FUNCTION_BLOCK ASSEMBLE_AD_FROM_AX (* this Function combines the 32 AX (BOOL) adapters to a AD (DWORD) *)
  (* Standard: 61499-2; Description: Copyright (c) 2026 Meisterschulen am Ostbahnhof SPDX-License-Identifier: EPL-2.0 *)
  (* Version 1.0, 2026-05-16, Franz Höpfinger, Meisterschulen am Ostbahnhof, initial API and implementation and/or initial documentation *)
  PACKAGE adapter::assembling;
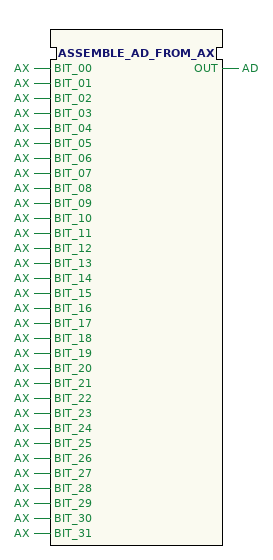
  SOCKETS
    BIT_00 : adapter::types::unidirectional::AX; (* Bool Bit 0 *)
    BIT_01 : adapter::types::unidirectional::AX; (* Bool Bit 1 *)
    BIT_02 : adapter::types::unidirectional::AX; (* Bool Bit 2 *)
    BIT_03 : adapter::types::unidirectional::AX; (* Bool Bit 3 *)
    BIT_04 : adapter::types::unidirectional::AX; (* Bool Bit 4 *)
    BIT_05 : adapter::types::unidirectional::AX; (* Bool Bit 5 *)
    BIT_06 : adapter::types::unidirectional::AX; (* Bool Bit 6 *)
    BIT_07 : adapter::types::unidirectional::AX; (* Bool Bit 7 *)
    BIT_08 : adapter::types::unidirectional::AX; (* Bool Bit 8 *)
    BIT_09 : adapter::types::unidirectional::AX; (* Bool Bit 9 *)
    BIT_10 : adapter::types::unidirectional::AX; (* Bool Bit 10 *)
    BIT_11 : adapter::types::unidirectional::AX; (* Bool Bit 11 *)
    BIT_12 : adapter::types::unidirectional::AX; (* Bool Bit 12 *)
    BIT_13 : adapter::types::unidirectional::AX; (* Bool Bit 13 *)
    BIT_14 : adapter::types::unidirectional::AX; (* Bool Bit 14 *)
    BIT_15 : adapter::types::unidirectional::AX; (* Bool Bit 15 *)
    BIT_16 : adapter::types::unidirectional::AX; (* Bool Bit 16 *)
    BIT_17 : adapter::types::unidirectional::AX; (* Bool Bit 17 *)
    BIT_18 : adapter::types::unidirectional::AX; (* Bool Bit 18 *)
    BIT_19 : adapter::types::unidirectional::AX; (* Bool Bit 19 *)
    BIT_20 : adapter::types::unidirectional::AX; (* Bool Bit 20 *)
    BIT_21 : adapter::types::unidirectional::AX; (* Bool Bit 21 *)
    BIT_22 : adapter::types::unidirectional::AX; (* Bool Bit 22 *)
    BIT_23 : adapter::types::unidirectional::AX; (* Bool Bit 23 *)
    BIT_24 : adapter::types::unidirectional::AX; (* Bool Bit 24 *)
    BIT_25 : adapter::types::unidirectional::AX; (* Bool Bit 25 *)
    BIT_26 : adapter::types::unidirectional::AX; (* Bool Bit 26 *)
    BIT_27 : adapter::types::unidirectional::AX; (* Bool Bit 27 *)
    BIT_28 : adapter::types::unidirectional::AX; (* Bool Bit 28 *)
    BIT_29 : adapter::types::unidirectional::AX; (* Bool Bit 29 *)
    BIT_30 : adapter::types::unidirectional::AX; (* Bool Bit 30 *)
    BIT_31 : adapter::types::unidirectional::AX; (* Bool Bit 31 *)
  END_SOCKETS
  PLUGS
    OUT : adapter::types::unidirectional::AD; (* DWORD Output *)
  END_PLUGS
  FBS
    ASSEMBLE_DWORD_FROM_BOOLS : eclipse4diac::utils::assembling::ASSEMBLE_DWORD_FROM_BOOLS;
    E_D_FF_ANY : iec61499::events::E_D_FF_ANY;
  END_FBS
  EVENT_CONNECTIONS
    BIT_00.E1 TO ASSEMBLE_DWORD_FROM_BOOLS.REQ;
    BIT_01.E1 TO ASSEMBLE_DWORD_FROM_BOOLS.REQ;
    BIT_02.E1 TO ASSEMBLE_DWORD_FROM_BOOLS.REQ;
    BIT_03.E1 TO ASSEMBLE_DWORD_FROM_BOOLS.REQ;
    BIT_04.E1 TO ASSEMBLE_DWORD_FROM_BOOLS.REQ;
    BIT_05.E1 TO ASSEMBLE_DWORD_FROM_BOOLS.REQ;
    BIT_06.E1 TO ASSEMBLE_DWORD_FROM_BOOLS.REQ;
    BIT_07.E1 TO ASSEMBLE_DWORD_FROM_BOOLS.REQ;
    BIT_08.E1 TO ASSEMBLE_DWORD_FROM_BOOLS.REQ;
    BIT_09.E1 TO ASSEMBLE_DWORD_FROM_BOOLS.REQ;
    BIT_10.E1 TO ASSEMBLE_DWORD_FROM_BOOLS.REQ;
    BIT_11.E1 TO ASSEMBLE_DWORD_FROM_BOOLS.REQ;
    BIT_12.E1 TO ASSEMBLE_DWORD_FROM_BOOLS.REQ;
    BIT_13.E1 TO ASSEMBLE_DWORD_FROM_BOOLS.REQ;
    BIT_14.E1 TO ASSEMBLE_DWORD_FROM_BOOLS.REQ;
    BIT_15.E1 TO ASSEMBLE_DWORD_FROM_BOOLS.REQ;
    BIT_16.E1 TO ASSEMBLE_DWORD_FROM_BOOLS.REQ;
    BIT_17.E1 TO ASSEMBLE_DWORD_FROM_BOOLS.REQ;
    BIT_18.E1 TO ASSEMBLE_DWORD_FROM_BOOLS.REQ;
    BIT_19.E1 TO ASSEMBLE_DWORD_FROM_BOOLS.REQ;
    BIT_20.E1 TO ASSEMBLE_DWORD_FROM_BOOLS.REQ;
    BIT_21.E1 TO ASSEMBLE_DWORD_FROM_BOOLS.REQ;
    BIT_22.E1 TO ASSEMBLE_DWORD_FROM_BOOLS.REQ;
    BIT_23.E1 TO ASSEMBLE_DWORD_FROM_BOOLS.REQ;
    BIT_24.E1 TO ASSEMBLE_DWORD_FROM_BOOLS.REQ;
    BIT_25.E1 TO ASSEMBLE_DWORD_FROM_BOOLS.REQ;
    BIT_26.E1 TO ASSEMBLE_DWORD_FROM_BOOLS.REQ;
    BIT_27.E1 TO ASSEMBLE_DWORD_FROM_BOOLS.REQ;
    BIT_28.E1 TO ASSEMBLE_DWORD_FROM_BOOLS.REQ;
    BIT_29.E1 TO ASSEMBLE_DWORD_FROM_BOOLS.REQ;
    BIT_30.E1 TO ASSEMBLE_DWORD_FROM_BOOLS.REQ;
    BIT_31.E1 TO ASSEMBLE_DWORD_FROM_BOOLS.REQ;
    ASSEMBLE_DWORD_FROM_BOOLS.CNF TO E_D_FF_ANY.CLK;
    E_D_FF_ANY.EO TO OUT.E1;
  END_CONNECTIONS
  DATA_CONNECTIONS
    ASSEMBLE_DWORD_FROM_BOOLS. TO E_D_FF_ANY.D;
    E_D_FF_ANY.Q TO OUT.D1;
    BIT_31.D1 TO ASSEMBLE_DWORD_FROM_BOOLS.BIT_31;
    BIT_30.D1 TO ASSEMBLE_DWORD_FROM_BOOLS.BIT_30;
    BIT_29.D1 TO ASSEMBLE_DWORD_FROM_BOOLS.BIT_29;
    BIT_28.D1 TO ASSEMBLE_DWORD_FROM_BOOLS.BIT_28;
    BIT_27.D1 TO ASSEMBLE_DWORD_FROM_BOOLS.BIT_27;
    BIT_26.D1 TO ASSEMBLE_DWORD_FROM_BOOLS.BIT_26;
    BIT_25.D1 TO ASSEMBLE_DWORD_FROM_BOOLS.BIT_25;
    BIT_24.D1 TO ASSEMBLE_DWORD_FROM_BOOLS.BIT_24;
    BIT_23.D1 TO ASSEMBLE_DWORD_FROM_BOOLS.BIT_23;
    BIT_22.D1 TO ASSEMBLE_DWORD_FROM_BOOLS.BIT_22;
    BIT_21.D1 TO ASSEMBLE_DWORD_FROM_BOOLS.BIT_21;
    BIT_20.D1 TO ASSEMBLE_DWORD_FROM_BOOLS.BIT_20;
    BIT_19.D1 TO ASSEMBLE_DWORD_FROM_BOOLS.BIT_19;
    BIT_18.D1 TO ASSEMBLE_DWORD_FROM_BOOLS.BIT_18;
    BIT_17.D1 TO ASSEMBLE_DWORD_FROM_BOOLS.BIT_17;
    BIT_16.D1 TO ASSEMBLE_DWORD_FROM_BOOLS.BIT_16;
    BIT_15.D1 TO ASSEMBLE_DWORD_FROM_BOOLS.BIT_15;
    BIT_14.D1 TO ASSEMBLE_DWORD_FROM_BOOLS.BIT_14;
    BIT_13.D1 TO ASSEMBLE_DWORD_FROM_BOOLS.BIT_13;
    BIT_12.D1 TO ASSEMBLE_DWORD_FROM_BOOLS.BIT_12;
    BIT_11.D1 TO ASSEMBLE_DWORD_FROM_BOOLS.BIT_11;
    BIT_10.D1 TO ASSEMBLE_DWORD_FROM_BOOLS.BIT_10;
    BIT_09.D1 TO ASSEMBLE_DWORD_FROM_BOOLS.BIT_09;
    BIT_08.D1 TO ASSEMBLE_DWORD_FROM_BOOLS.BIT_08;
    BIT_07.D1 TO ASSEMBLE_DWORD_FROM_BOOLS.BIT_07;
    BIT_06.D1 TO ASSEMBLE_DWORD_FROM_BOOLS.BIT_06;
    BIT_05.D1 TO ASSEMBLE_DWORD_FROM_BOOLS.BIT_05;
    BIT_04.D1 TO ASSEMBLE_DWORD_FROM_BOOLS.BIT_04;
    BIT_03.D1 TO ASSEMBLE_DWORD_FROM_BOOLS.BIT_03;
    BIT_02.D1 TO ASSEMBLE_DWORD_FROM_BOOLS.BIT_02;
    BIT_01.D1 TO ASSEMBLE_DWORD_FROM_BOOLS.BIT_01;
    BIT_00.D1 TO ASSEMBLE_DWORD_FROM_BOOLS.BIT_00;
  END_CONNECTIONS
END_FUNCTION_BLOCK
